// TIA Portal V20 export
FUNCTION "SysCal1x" : Void   // FC2010, FBD
TITLE = one point callibration, work only with encoder data structure
{ S7_Optimized_Access := 'TRUE' }
AUTHOR : MiCROTEC
VERSION : 1.0
// -2017.03 : Martin
// stored: AutoNumber false, SetENOAutomatically false
   VAR_INPUT
      p1Set : Bool;   // set calibration point 1
      p1Inc : DInt;   // callibration point 1 in increment
      p1Mm : Real;   // callibration point 1 in millimeter
      encAct : DInt;   // actual position encoder
      gain : Real;   // callibration gain
      limMin : Real;   // limit position minimum
      limMax : Real;   // limit position maximum
      ack : Bool;   // fault acknowledge
   END_VAR
   VAR_OUTPUT
      calGain : Real;   // callibration gain
      calOffset : Real;   // callibration offset
      act : Real;   // actual position
      err : Bool;   // fault
   END_VAR
   VAR_IN_OUT
      Enc : "TypeEncoder";
   END_VAR
   VAR_TEMP
      tempAct : Real;   // actual position
   END_VAR
BEGIN

REGION Network 1: save callibration point 1
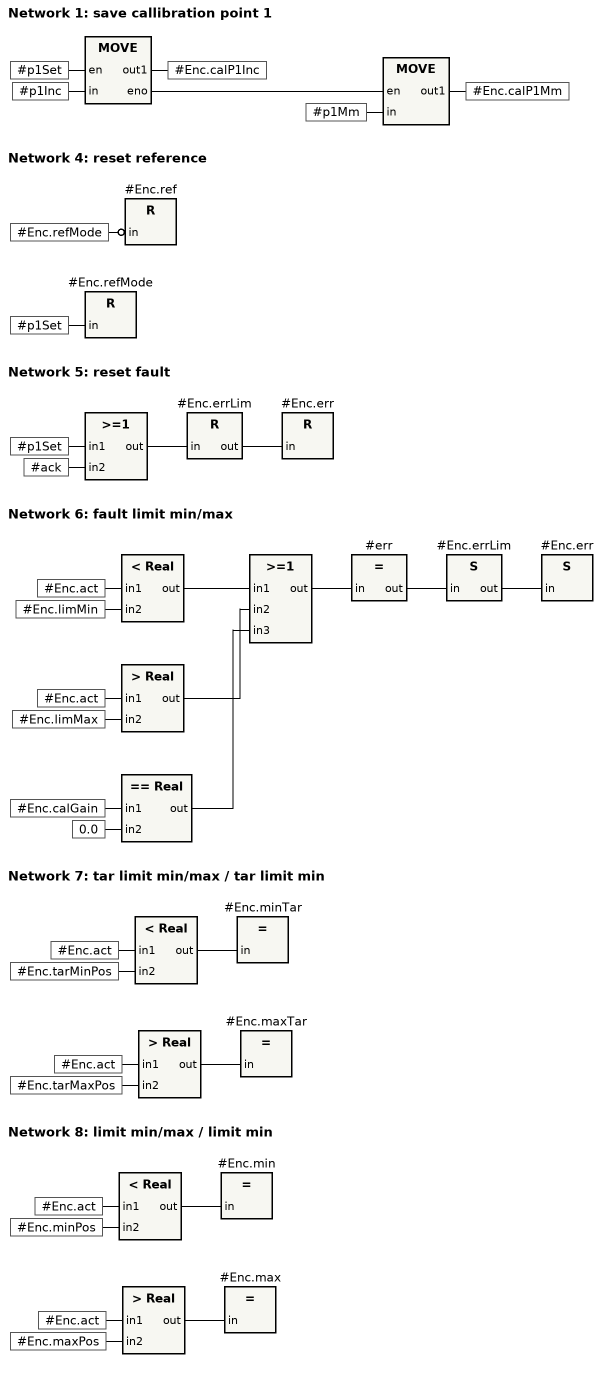
   // ENO of a box is taken as its EN; it also drops when the box reports an error
   IF #p1Set THEN
       #Enc.calP1Inc := #p1Inc;
       #Enc.calP1Mm := #p1Mm;
   END_IF;
END_REGION

REGION Network 2 (SCL): calculations
   #Enc.calGain := #gain;
   #Enc.calOffset := #Enc.calP1Mm - (DINT_TO_REAL(#Enc.calP1Inc) * #Enc.calGain);

   #Enc.act := (DINT_TO_REAL(#encAct - #Enc.calP1Inc) * #Enc.calGain) + #Enc.calP1Mm;
   #Enc.delta := DINT_TO_REAL(#Enc.deltaInc) * #Enc.calGain;
   #Enc.speed := #Enc.delta * 60.0 / "cycle";
END_REGION

REGION Network 3 (SCL): read/write values
   #Enc.limMin := #limMin;
   #Enc.limMax := #limMax;

   #calOffset := #Enc.calOffset;
   #calGain := #Enc.calGain;
   #act := #Enc.act;
END_REGION

REGION Network 4: reset reference
   IF NOT #Enc.refMode THEN #Enc.ref := FALSE; END_IF;
   IF #p1Set THEN #Enc.refMode := FALSE; END_IF;
END_REGION

REGION Network 5: reset fault
   IF #p1Set OR #ack THEN
       #Enc.errLim := FALSE;
       #Enc.err := FALSE;
   END_IF;
END_REGION

REGION Network 6: fault limit min/max
   #err := (#Enc.act < #Enc.limMin) OR (#Enc.act > #Enc.limMax) OR (#Enc.calGain = 0.0);
   IF #err THEN
       #Enc.errLim := TRUE;
       #Enc.err := TRUE;
   END_IF;
END_REGION

REGION Network 7: tar limit min/max / tar limit min
   #Enc.minTar := #Enc.act < #Enc.tarMinPos;
   #Enc.maxTar := #Enc.act > #Enc.tarMaxPos;
END_REGION

REGION Network 8: limit min/max / limit min
   #Enc.min := #Enc.act < #Enc.minPos;
   #Enc.max := #Enc.act > #Enc.maxPos;
END_REGION
END_FUNCTION
